GLOBALCONSTANTS AID_WM (* Window mask object attribute ids *)
  (* Standard: 61499-1; Description: Copyright (c) 2023 HR Agrartechnik GmbH This program and the accompanying materials are made available under the terms of the Eclipse Public License 2.0 which is available at https://www.eclipse.org/legal/epl-2.0/ SPDX-License-Identifier: EPL-2.0 *)
  (* Version 1.0, 2026-06-20, Franz Höpfinger, HR Agrartechnik GmbH *)
  PACKAGE isobus::UT::Q::const::AID;
  IMPORT eclipse4diac::core::TypeHash;
  VAR_GLOBAL CONSTANT
    BACKGROUND_COLOUR : USINT := USINT#1; (* 1: AID_WM_BACKGROUND_COLOUR - Background colour index. *)
    OPTIONS : USINT := USINT#2; (* 2: AID_WM_OPTIONS - Bitmask: Bit 0 = Available (0=disable/blank window), Bit 1 = Transparent (no background colour). *)
    NAME : USINT := USINT#3; (* 3: AID_WM_NAME - Object ID of an Output String or Object Pointer containing the name. *)
  END_VAR
END_GLOBALCONSTANTS
